Staubli VAL3: INT_EDIT.pgx

program Int_Edit(num& x_nData, num x_nX, num x_nY)
  local num l_nKey
  local num l_nNum
begin
  //说明：
  //函数功能：在划定的框内，对数值类型变量进行编辑


  call Int_EditS(x_nData,x_nX,x_nY,"")
end
